Staubli VAL3: page_simulation.pjx

--- page_simulation.pjx ---
Parameters version=s7.8.3 stackSize=5000 millimeterUnit=true
Program file=CycleRefresh.pgx
Program file=goTo.pgx
Program file=isAtPoint.pgx
Program file=loadEditTraj.pgx
Program file=loadPage.pgx
Program file=loadType.pgx
Program file=main.pgx
Program file=onEnterEvent.pgx
Program file=onExit.pgx
Program file=onF1Event.pgx
Program file=onF2Event.pgx
Program file=onF3Event.pgx
Program file=onF4Event.pgx
Program file=onF5Event.pgx
Program file=onF6Event.pgx
Program file=onF7Event.pgx
Program file=onF8Event.pgx
Program file=onStart.pgx
Program file=printToShow.pgx
Program file=refresh.pgx
Program file=refreshDynamic.pgx
Program file=refreshPoints.pgx
Program file=refreshStatic.pgx
Program file=showMessage.pgx
Program file=startCycle.pgx
Program file=stepping.pgx
Program file=stopCycle.pgx
Data file=page_simulation.dtx
Library alias=page path=Disk://kernel/template/page/page.pjx
Library alias=use path=Disk://kernel/userPage/userPage.pjx
Library alias=language path=Disk://kernel/language/language.pjx
Library alias=saveData path=Disk://saveData/saveData.pjx
Library alias=cycleStatus path=Disk://cycleStatus/cycleStatus.pjx
Library alias=trajType path=Disk://../templates/trajectory/trajectory.pjx
Library alias=OnEvent path=Disk://OnEvent/OnEvent.pjx

--- page_simulation.dtx ---
num nEvent
num nIndex
num nKey
public num nPage
num nPoint
num nRefresh = 1
num nSelect
num nTime = 1.5
public num nToSuperV
num nRoundStepping = 25
num nMoveId
string sEvent
public string sItems
string sList
string sMenu
string sMessage
string sTrajName
string sMenu8[8]
bool bButton[8]
bool bMoveToPoint
bool bShowMessage
bool bShowStatus
bool bStepping
mdesc nom_speed = {accel=50, vel=50, decel=50, tmax=999, rmax=999, blend=off}

--- main.pgx ---
public program main()
  local num i
  local num l_nResult
begin
  cls()
  // INIT
  call onStart(l_nResult)
  //
  //
  if trajType:bStepping
    if l_nResult==0
      // LOOP UNTIL nKey=255
      do
        //
        nKey=getKey()
        // REFRESH
        call refresh()
        //
        switch nKey
          case 271 ,264
            // previous
            call onF1Event()
          break
          case 272
            // actual
            call onF2Event()
          break
          case 273 ,268
            // next
            call onF3Event()
          break
          case 274
            call onF4Event()
          break
          case 275
            call onF5Event()
          break
          case 276
            call onF6Event()
          break
          case 277,255
            call onF7Event()
          break
          case 278
            call onF8Event()
          break
          case 270
            call onEnterEvent()
          break
        endSwitch
        // release
        delay(0)
      until nKey==255
      // on Exit
      call onExit()
    else
      //
      // check
      //
      popUpMsg("ERROR..: "+toString("",l_nResult))
      logMsg("ERROR loading, "+toString("",l_nResult))
    endIf
    //
  endIf
end

--- CycleRefresh.pgx ---
program CycleRefresh()
  local num l_nEvent
  local num l_nSize[3]
  local num i
  local num l_nResult
  local bool l_bTrajRunning
begin
  // set the size
  call use:setSizeList(19,0,19,10)
  //
  // TRAJECTORY
  //
  if use:bUseRefresh
    // refresh the board
    call refreshStatic()
    //
    use:bUseRefresh=false
    //
    // rebuilt the Traj list
    //
    call refreshPoints(saveData:sTrajTypeUsing+" "+sTrajName)
    // look if the init has finished
    if cycleStatus:bSimulation
      nPoint=cycleStatus:nPoint
    endIf
    // REFRESH ACTUAL POINT
    use:nView=nPoint%use:nBottomY
    call use:listredraw(nPoint-use:nView)
  else
    // only update
    nPoint=cycleStatus:nPoint
    if use:nView>=nPoint%use:nBottomY
      // update the list
      use:nView=nPoint%use:nBottomY
      call use:listupdate(nPoint-use:nView)
    else
      //just the line
      call use:listcursor(use:nView,false)
      use:nView=nPoint%use:nBottomY
      call use:listcursor(use:nView,true)
    endIf
  endIf
end

--- goTo.pgx ---
program goTo(num x_nIndex)
  local string l_sActualTraj
  local tool l_tTool
  local bool l_bUnreached
  local string l_sMessage
  local num i
  local bool l_bContinue
  local num l_nIndexTool
  local bool l_bInside
  local bool l_bSamePoint
  local num l_nSize
  local num l_nTcpAction
  local string l_sEmpty
  local num l_nZero
  local TrajectoryItem l_tItem
begin
  // clean the movement
  if !isEmpty()
    resetMotion()
  endIf
  // get the tcp
  call trajType:getTool(l_nIndexTool)
  call saveData:getTool(l_tTool,l_nIndexTool)
  // get the trajType
  call trajType:getTrajItem(l_tItem,x_nIndex)
  // set the blend to off
  l_tItem.nom_speed.blend=off
  // AUTO ON
  if cycleStatus:nWorkingMode!=1
    // put the auto ON
    cycleStatus:bAutoON=true
    if watch(cycleStatus:bAutoON==false,3)
      l_bContinue=true
    endIf
  else
    l_bContinue=true
  endIf
  if l_bContinue
    //
    cls()
    // goTO
    call trajType:goTo(l_tTool,l_tItem.nom_speed,l_tItem.moveType,l_bUnreached,x_nIndex)
    if l_bUnreached
      // ERROR POINT NOT REACHABLE
      call language:message(l_sMessage,-5)
      call use:timerDialog(l_sMessage,1)
    else
      // GO ON
      do
        // refresh the scroll bar
        nMoveId=getMoveId()
        call use:type(0,11,toString("2",nPoint+1)+" ")
        call use:type(37,11,toString("2",x_nIndex+1)+" ")
        call use:scroll(3,11,32,abs(roundDown(nMoveId)-nMoveId)*100)
        // move to the point
        bMoveToPoint=true
        call use:typeMenu(7,"STOP")
        call showMessage()
        if !bShowMessage
          call language:message(l_sMessage,94)
          call use:timerDialog(l_sMessage+toString("",x_nIndex+1),0)
        endIf
        //
        nKey=getKey()
        delay(0)
      until (isEmpty() or nKey==255 or nKey==277)
    endIf
    //
    //look if the robot has moved
    call isAtPoint(nPoint,l_bInside)
    //DEBUT MODIF A VALIDER
    call trajType:getSizeItem(false,l_nSize)
    if nPoint<l_nSize-1
      call isAtPoint(nPoint+1,l_bSamePoint)
    endIf
    //FIN MODIF A VALIDER (+ le or l_bSamePoint)
    if !l_bInside and nPoint<x_nIndex or l_bSamePoint
      //update the nPoint
      nPoint=x_nIndex
    else
      // back position
      call isAtPoint(x_nIndex,l_bInside)
      if l_bInside and nPoint>x_nIndex
        // update the point
        nPoint=x_nIndex
      endIf
    endIf
    resetMotion()
    //
    use:bUseRefresh=true
    // clean
    bMoveToPoint=false
    call use:nullKey(nKey)
  endIf
end

--- onExit.pgx ---
program onExit()
begin
  // on EXIT
  //
  if cycleStatus:bSimulation
    call stopCycle()
  endIf
  // clean the movement
  if !isEmpty()
    resetMotion()
  endIf
  call use:nullKey(nKey)
  taskKill("stepping")
end

--- onF3Event.pgx ---
program onF3Event()
  local string l_sMessage
  local bool l_bInside
begin
  // look if the bButton is enable
  if bButton[2]
    //
    // go to next POINT
    //
    if !cycleStatus:bCycle or !cycleStatus:bSimulation
      // check for the point proximity
      call isAtPoint(nPoint,l_bInside)
      if l_bInside
        call goTo(nPoint+1)
      else
        call goTo(nPoint)
      endIf
    endIf
  endIf
end

--- onF4Event.pgx ---
program onF4Event()
begin
  // look if the bButton is enable
  if bButton[3]
    //
    //
    //
  endIf
end

--- onF6Event.pgx ---
program onF6Event()
  local num l_nSize
begin
  // look if the bButton is enable
  if bButton[5]
   //
    if cycleStatus:bSimulation and cycleStatus:bPause and esStatus()!=2
      call OnEvent:resumeCycle()
    endIf
  endIf
end

--- onF8Event.pgx ---
program onF8Event()
  local string l_sMessage
begin
  // look if the bButton is enable
  if bButton[7]
    //
  endIf
end

--- printToShow.pgx ---
program printToShow()
  local num l_nSize
  local string l_sMessage
  local num l_nScrool
  local bool l_bInside
begin
  //
  //  Print the instruction and the function KEY STEP
  //
  call use:typeLen(0,12,""+cycleStatus:sToShow,40)
  //
  // refresh the scroll bar in simulation
  //
  if cycleStatus:bSimulation
    nMoveId=getMoveId()
  endIf
  if nMoveId>=1
    call trajType:getSizeItem(false,l_nSize)
    // normal point
    call use:type(0,11,toString("2",nPoint)+" ")
    call use:type(37,11,toString("2",nPoint+1)+" ")
  else
    // start Point
    call use:type(0,11,toString("2",nPoint)+" ")
    call use:type(37,11,toString("2",nPoint+1)+" ")
  endIf
  // print the scroll
  call isAtPoint(nPoint,l_bInside)
  if l_bInside
    l_nScrool=100
  else
    l_nScrool=abs(roundDown(nMoveId)-nMoveId)*100
  endIf
  call use:scroll(3,11,32,l_nScrool)
  call language:message(l_sMessage,124)
end

--- refresh.pgx ---
program refresh()
// // page refresh
  local string l_sMessage
begin
  if !bShowMessage
    if (nKey>=270 and nKey<=278) or abs(clock()-nRefresh)>nTime
      // refresh the static message
      use:bUseRefresh=true
      call refreshDynamic()
    else
      // refresh the Dynamic message
      if use:bUseRefresh
        call refreshDynamic()
      endIf
    endIf
  endIf
  // show the message
  call showMessage()
  // print the instruction
  call printToShow()
end

--- refreshDynamic.pgx ---
program refreshDynamic()
begin
  // DO NOT CHANGE
  nRefresh=clock()
  //
  // ADD HERE
  //
  call CycleRefresh()
  //
  use:bUseRefresh=false
end

--- refreshStatic.pgx ---
program refreshStatic()
  local string l_sMenu
  local string l_sMessage
  local num i
  local num l_nSize
  local bool l_bInside
begin
  //
  // set the view of the page..
  //
  // SET THE PAGE NUMBER
  // clean the left Side
  for i=0 to 10
    call use:typeLen(0,i," ",19)
  endFor
  use:nPage=210
  // USE <>PROFILE for <>PAGE
  use:nPage=use:nPage+abs(limit(saveData:mode,0,2)-2)
  if cycleStatus:bCycle
    use:nPage=use:nPage+3
  endIf
  // load the menu page
  if saveData:language!="japanese"
    // SET THE VIEW OF THE PAGE
    call language:page(l_sMessage,use:nPage)
    // define the menu
    call use:stringToArray(l_sMessage,sMenu)
  else
    // japanese use the array for the menu
    call language:page(sMenu8,use:nPage)
    call use:stringCopy(sMenu8,sMenu)
  endIf
  //
  // set the menu
  call use:clear(0,13)
  call trajType:getSizeItem(false,l_nSize)
  //
  //
  if !cycleStatus:bSimulation
    //
    // NOT IN CYCLE
    //
    // CHANGE ICON
    // CHECK THE INDEX
    // check for the point proximity
    call isAtPoint(nPoint,l_bInside)
    if l_bInside
      sMenu[1]=""
    else
      // clean it
      sMenu[2]=""
    endIf
    // start
    if nPoint<=0
      // previous
      sMenu[0]=""
    endIf
    if nPoint>=l_nSize-1
      // clean it
      sMenu[2]=""
    endIf
    // START
    call use:type(31,13,"START")
  else
    //
    // IN CYCLE
    //
    // STOP
    call use:type(31,13,"STOP ")
    if cycleStatus:bPause
      call use:type(24,13,"RESTART")
    else
      call use:type(24,13,"       ")
    endIf
    // disable << X >>
    sMenu[0]=""
    sMenu[1]=""
    sMenu[2]=""
    sMenu[3]=""
  endIf
  // set the menu
  if saveData:language!="japanese"
    call use:setMenu(sMenu,true,3)
  else
    call use:setMenu(sMenu,false,3)
  endIf
  call use:getMenu(sMenu,bButton)
  if !cycleStatus:bSimulation
    call isAtPoint(nPoint,l_bInside)
    if !l_bInside
      // actual
      call use:typeMenu(2,"X")
    elseIf nPoint<l_nSize-1
      // next
      call use:typeMenu(3,">>")
    endIf
    if nPoint>0
      // previuos
      call use:typeMenu(1,"<<")
    endIf
    // look for the STEP ENABLING
  elseIf !bStepping and nPoint<(l_nSize-1) and nPoint>0 and taskStatus("stepping")==-1 and !isEmpty()
    call use:typeMenu(2,"STEP")
    bButton[1]=true
  endIf
  call language:message(l_sMessage,124)
  // START STOP
  bButton[6]=true
  //
end

--- showMessage.pgx ---
program showMessage()
  local string l_sMessage
begin
  // INIT
  bShowMessage=false
  // look for the esStatus
  if esStatus()==2
    call language:message(l_sMessage,222)
    bShowMessage=true
  else
    // look for the Working Mode and power in SimulMode
    if cycleStatus:bSimulation or bMoveToPoint
      if !isPowered() and cycleStatus:nWorkingMode!=4
        call language:message(l_sMessage,201)
        bShowMessage=true
      elseIf cycleStatus:nWorkingStatus!=0
        // PRESS MOVE HOLD
        call language:message(l_sMessage,203)
        if cycleStatus:nWorkingMode==1
          switch cycleStatus:nWorkingStatus
            case 2
              // JOINT
              call language:message(l_sMessage,140)
            break
            case 3
              // WORLD
              call language:message(l_sMessage,141)
            break
            case 4
              // TOOL
              call language:message(l_sMessage,142)
            break
            case 5
              // POINT
              call language:message(l_sMessage,143)
            break
          endSwitch
        endIf
        bShowMessage=true
      elseIf bStepping
        l_sMessage=" STEPPING ..."
        bShowMessage=true
      endIf
    endIf
  endIf
  //
  if bShowMessage
    call use:timerDialog(l_sMessage,0)
  endIf
end
